// TwinCAT 3 PLC project Fs_Standard
// Title: FisoThemes Standard Library
// Company: FisoThemes
// ProjectVersion: 0.0.0.0
// ProgramVersion: 3.1.4023.0
// libraries:
//   Tc2_Standard, * (Beckhoff Automation GmbH)
//   Tc2_System, * (Beckhoff Automation GmbH)
//   Tc3_Module, * (Beckhoff Automation GmbH)
// project tree:
//   Core/DataUnitTypes/Alias/ FsT_Accessor.TcDUT, FsT_Char.TcDUT, FsT_SStr.TcDUT, FsT_MemArea.TcDUT, FsT_PlcAppInfo.TcDUT, FsT_PlcTaskInfo.TcDUT, FsT_Ptr.TcDUT, FsT_Size.TcDUT, FsT_Str.TcDUT, FsT_LStr.TcDUT, FsT_TypeClass.TcDUT, FsT_VarInfo.TcDUT
//   Core/DataUnitTypes/Enums/ FsE_Accessor.TcDUT
//   Core/DataUnitTypes/Structs/ FsST_PlcTaskInformation.TcDUT
//   Core/FunctionBlocks/ FsFB_Object.TcPOU, FsFB_ValueType.TcPOU
//   Core/Functions/ FsF_Cast.TcPOU, FsF_GetAddress.TcPOU, FsF_GetSize.TcPOU, FsF_GetPlcTaskInformation.TcPOU, FsF_GetTypeNameByAddress.TcPOU, FsF_GetTypeName.TcPOU, FsF_GetVariablePathByAddress.TcPOU, FsF_GetTypeNameByPath.TcPOU, FsF_GetVariablePath.TcPOU
//   Core/Interfaces/ FsI_Cloneable.TcIO, FsI_Equatable.TcIO, FsI_Unknown.TcIO, FsI_Object.TcIO, FsI_ValueType.TcIO
//   Core/Parameters/ FsParam_Core.TcGVL
//   Core/_Playground/ FsP_CorePlayground.TcPOU
//   ErrorHandling/DataUnitTypes/Alias/ FsT_ErrMsg.TcDUT, FsT_ErrSrc.TcDUT, FsT_ErrCode.TcDUT
//   ErrorHandling/FunctionBlocks/ FsFB_Error.TcPOU, FsFB_ErrorDefinition.TcPOU, FsFB_ErrorDefinitionOnInit.TcPOU
//   ErrorHandling/Functions/ FsF_Error.TcPOU, FsF_ErrorPath.TcPOU
//   ErrorHandling/Globals/ FsGVL_CodesysCmpErrors.TcGVL, FsGVL_ErrorCodes.TcGVL
//   ErrorHandling/Interfaces/ FsI_Error.TcIO
//   ErrorHandling/Parameters/ FsParam_ErrorHandling.TcGVL
//   / PlcTask.TcTTO
//   Project Information/ F_GetCompany.TcPOU, F_GetTitle.TcPOU, F_GetVersion.TcPOU
//   Version/ Global_Version.TcGVL
//   _Internal/FunctionBlocks/ FsFB_TcComIecApplicationInfo.TcPOU
//   _Internal/Globals/ _FsGVL.TcGVL
//   _Internal/ _MAIN.TcPOU
//   _TemplateFolder/_Playground/ FsP_TempPlayground.TcPOU
//   ErrorHandling/_Playground/ FsP_ErrorHandlingPlayground.TcPOU
// real-time tasks:
//   TASK PlcTask: cycle T#1ms, priority 20, ADS port 350

CONFIGURATION Fs_Standard
    RESOURCE PLC ON TwinCAT3
        TASK PlcTask(INTERVAL := T#1ms, PRIORITY := 20);
        PROGRAM _MAIN WITH PlcTask : _MAIN;
        PROGRAM FsP_CorePlayground WITH PlcTask : FsP_CorePlayground;
        PROGRAM FsP_ErrorHandlingPlayground WITH PlcTask : FsP_ErrorHandlingPlayground;
    END_RESOURCE
END_CONFIGURATION

// ---- Core/DataUnitTypes/Alias/FsT_Accessor.TcDUT
// An enum that can be used to represent getters and setters.
TYPE FsT_Accessor : FsE_Accessor; END_TYPE

// ---- Core/DataUnitTypes/Alias/FsT_Char.TcDUT
// Single character string.
TYPE FsT_Char : STRING(1); END_TYPE

// ---- Core/DataUnitTypes/Alias/FsT_SStr.TcDUT
// Short string.
// Size is a parameter located at FSParam_Core.nFST_SSTR_SIZE. | DEFAULT: 40
TYPE FsT_SStr : STRING(FSParam_Core.SSTR_SIZE); END_TYPE

// ---- Core/DataUnitTypes/Alias/FsT_MemArea.TcDUT
TYPE FsT_MemArea : Tc2_System.E_TcMemoryArea; END_TYPE

// ---- Core/DataUnitTypes/Alias/FsT_PlcAppInfo.TcDUT
TYPE FsT_PlcAppInfo : PlcAppSystemInfo; END_TYPE

// ---- Core/DataUnitTypes/Alias/FsT_PlcTaskInfo.TcDUT
TYPE FsT_PlcTaskInfo : FsST_PlcTaskInformation; END_TYPE

// ---- Core/DataUnitTypes/Alias/FsT_Ptr.TcDUT
TYPE FsT_Ptr : POINTER TO BYTE; END_TYPE

// ---- Core/DataUnitTypes/Alias/FsT_Size.TcDUT
TYPE FsT_Size : UXINT; END_TYPE

// ---- Core/DataUnitTypes/Alias/FsT_Str.TcDUT
// Standard FS string.
// Size is a parameter located at FSParam_Core.nFST_STR_SIZE. | DEFAULT: 80
TYPE FsT_Str : STRING(FSParam_Core.STR_SIZE); END_TYPE

// ---- Core/DataUnitTypes/Alias/FsT_LStr.TcDUT
// Long string.
// Size is a parameter located at FSParam_Core.nFST_STR_SIZE. | DEFAULT: 80
TYPE FsT_LStr : STRING(FSParam_Core.LSTR_SIZE); END_TYPE

// ---- Core/DataUnitTypes/Alias/FsT_TypeClass.TcDUT
TYPE FsT_TypeClass : __SYSTEM.TYPE_CLASS; END_TYPE

// ---- Core/DataUnitTypes/Alias/FsT_VarInfo.TcDUT
TYPE FsT_VarInfo : __SYSTEM.VAR_INFO; END_TYPE

// ---- Core/DataUnitTypes/Enums/FsE_Accessor.TcDUT
// An enum that can be used to represent getters and setters.
{attribute 'qualified_only'}
{attribute 'strict'}
{attribute 'to_string'}
TYPE FsE_Accessor :
(
	_ := 0,
	Get,
	Set
);
END_TYPE

// ---- Core/DataUnitTypes/Structs/FsST_PlcTaskInformation.TcDUT
TYPE FsST_PlcTaskInformation :
STRUCT
	 ObjId                   : OTCID; // Object ID of the task reference, from which the PLC program is called.
     CycleTime               : LTIME; // Task cycle time.
     Priority                : UINT; // Task priority.
     AdsPort                 : UINT; // Task ADS port.
     CycleCount              : UDINT; // Cycle counter. | NOTE: This refers to the actual system task and not to the task reference of the PLC project.
     DcTaskTime              : LINT; // Distributed Clock System Time. | NOTE: It remains constant for a task runtime.
     LastExecTime            : LTIME; // Cycle time required for the last cycle.
     FirstCycle              : BOOL; // During the first PLC task cycle, this variable has the value TRUE.
     CycleTimeExceeded       : BOOL; // Indicates whether the set task cycle time was exceeded.
     InCallAfterOutputUpdate : BOOL; // This TRUE if the origin of the current call is declared with the attribute 'TcCallAfterOutputUpdate'.
     RTViolation             : BOOL; // This variable has the value TRUE if the real-time limit is exceeded on a mixed core (Windows + real-time on one core).
     TaskName                : STRING(63); // Name of the task reference object in the PLC project (e.g. 'MyPlcProject_PlcTaskRef')
	 TaskIndex 				 : BYTE; // Task index of the task.
END_STRUCT
END_TYPE

// ---- ErrorHandling/DataUnitTypes/Alias/FsT_ErrMsg.TcDUT
TYPE FsT_ErrMsg : STRING(FsParam_ErrorHandling.ERROR_MSG_SIZE); END_TYPE

// ---- ErrorHandling/DataUnitTypes/Alias/FsT_ErrSrc.TcDUT
TYPE FsT_ErrSrc : STRING(FsParam_ErrorHandling.ERROR_SRC_SIZE); END_TYPE

// ---- ErrorHandling/DataUnitTypes/Alias/FsT_ErrCode.TcDUT
TYPE FsT_ErrCode : LINT; END_TYPE

// ---- Core/Parameters/FsParam_Core.TcGVL
{attribute 'qualified_only'}
VAR_GLOBAL CONSTANT
	STR_SIZE : FsT_Size := 80; // Size of general string.
	SSTR_SIZE : FsT_Size := 40; // Size of short string.
	LSTR_SIZE : FsT_Size := 255; // Size of long string.
	INFO_SCAN_SIZE : FsT_Size := 15000; // How many bytes to scan when looking for information. e.g. it's FsFB_Object to find the size of a child object in static memory.
END_VAR

// ---- ErrorHandling/Globals/FsGVL_CodesysCmpErrors.TcGVL
{attribute 'qualified_only'}
(* Error code are @ CmpErrors.Errors.<variable> from the CmpErrors2 Interfaces library.*)
VAR_GLOBAL CONSTANT
	ERR_OK 						: FsT_ErrCode := 16#0; 		//	Ok
	ERR_FAILED 					: FsT_ErrCode := 16#1; 		//	General error - To be used only for internal errors
	ERR_PARAMETER 				: FsT_ErrCode := 16#2; 		//	Invalid parameter for this operation
	ERR_NOTINITIALIZED 			: FsT_ErrCode := 16#3; 		//	Function cannot be executed, since component has not been initialized yet. It may work later, though
	ERR_VERSION 				: FsT_ErrCode := 16#4; 		//	Version conflict
	ERR_TIMEOUT 				: FsT_ErrCode := 16#5; 		//	Operation timed out
	ERR_NOBUFFER 				: FsT_ErrCode := 16#6; 		//	Insufficient memory to carry out the request
	ERR_PENDING 				: FsT_ErrCode := 16#A; 		//	For async-calls: call not complete, yet
	ERR_NUMPENDING 				: FsT_ErrCode := 16#B; 		//  Too many pending calls. Try later
	ERR_NOTIMPLEMENTED 			: FsT_ErrCode := 16#C; 		//  The function is not implemented
	ERR_INVALIDID 				: FsT_ErrCode := 16#D; 		//  No object with the provided id found
	ERR_OVERFLOW 				: FsT_ErrCode := 16#E; 		//	Integer overflow
	ERR_BUFFERSIZE 				: FsT_ErrCode := 16#F; 		//	The size of a buffer is too small OR invalid
	ERR_NO_OBJECT 				: FsT_ErrCode := 16#10;		//	No object with THIS specified name available
	ERR_NOMEMORY 				: FsT_ErrCode := 16#11;		//  No heap memory available
	ERR_DUPLICATE 				: FsT_ErrCode := 16#12A;  	//  An object with the same name is still available
	ERR_MEMORY_OVERWRITE 		: FsT_ErrCode := 16#13;  	//  Heap memory was written out of bounds! Memory overwrite error
	ERR_INVALID_HANDLE 			: FsT_ErrCode := 16#14;  	//  Invalid handle to an object
	ERR_END_OF_0BJECT 			: FsT_ErrCode := 16#15;  	//  End OF object reached
	ERR_NO_CHANGE 				: FsT_ErrCode := 16#16;  	//  No changes done
	ERR_INVALID_INTERFACE 		: FsT_ErrCode := 16#17;  	//  Invalid OR unknown interface
	ERR_NOT_SUPPORTED 			: FsT_ErrCode := 16#18;  	//  Functionality not supported
	ERR_NO_ACCESS_RIGHTS 		: FsT_ErrCode := 16#19;  	//  No access rights for this operation
	ERR_OUT_OF_LIMITS 			: FsT_ErrCode := 16#1A;  	//  Specified limits of a resource exceeded
	ERR_ENTRIES_REMAINING 		: FsT_ErrCode := 16#18;  	//  Remaining entries that could not be transmitted because of buffer limitation
	ERR_INVALID_SESSION_ID 		: FsT_ErrCode := 16#1C;  	//  Invalid online sessionid
	ERR_EXCEPTION 				: FsT_ErrCode := 16#1D;  	//  Exception occurred
	ERR_SIGNATURE_MISMATCH 		: FsT_ErrCode := 16#1E;		//	Signature mismatch of an api function
	ERR_VERSION_MISMATCH 		: FsT_ErrCode := 16#1F;		//	Version mismatch
	ERR_TYPE_MISMATCH 			: FsT_ErrCode := 16#20;		//	Type mismatch
	ERR_ID_MISMATCH 			: FsT_ErrCode := 16#21;		//	ID mismatch
	ERR_NO_CONSISTENCY 			: FsT_ErrCode := 16#22;		//	Consistency error
	ERR_NO_COMM_CYCLE 			: FsT_ErrCode := 16#23;		//	No COMM_CYCLE needed
	ERR_DONT_SUSPEND_TASK 		: FsT_ErrCode := 16#24;		//	Do not suspend task after an exception
	ERR_MEMORY_LOCK_FAILED 		: FsT_ErrCode := 16#25;		//	Memory cannot be locked in this operation
	ERR_LICENSE_MISSING 		: FsT_ErrCode := 16#26;		//	License missing for the runtime
	ERR_OPERATION_DENIED 		: FsT_ErrCode := 16#27;		//	Operation denied 
	ERR_DEVICE 					: FsT_ErrCode := 16#28;		//	Device error
	ERR_DISK_FULL 				: FsT_ErrCode := 16#29;		//	Disk full
	ERR_CRC_FAILED 				: FsT_ErrCode := 16#30;		//	Internal use in runtime
	ERR_MEDIA_ERASE 			: FsT_ErrCode := 16#31;		//	Internal use in runtime
	ERR_FILE_ERROR 				: FsT_ErrCode := 16#32;		//	File error. e.g. cannot open a file for writing because it could be write protected
	ERR_NO_RETAIN_MEMORY 		: FsT_ErrCode := 16#33;		//	No retain memory available
	ERR_OUT_OF_LIMITS_MIN 		: FsT_ErrCode := 16#34;		//	Specified minimum-limit of a resource exceeded
	ERR_OUT_OF_LIMITS_MAX 		: FsT_ErrCode := 16#35;		//	Specified maximum-limit of a resource exceeded
	ERR_SIZE_MISMATCH 			: FsT_ErrCode := 16#36;		//	Size mismatch
	ERR_CALL_AGAIN 				: FsT_ErrCode := 16#37;		//	Operation is not yet finished, call function again to proceed
	ERR_NOTHING_TO_DO 			: FsT_ErrCode := 16#38;		//	Operation has nothing to do. No execution.
	ERR_SECURITY_CHECKS_FAILED 	: FsT_ErrCode := 16#39;		//	Some security checks have failed. /* This is a generic error code to report this error over public channels. In this case the error code doesn’t provide a detailed cause for the error. */
	ERR_INVALID_SEQUENCE 		: FsT_ErrCode := 16#3A;		//	 
	ERR_INVALID_REFERENCE 		: FsT_ErrCode := 16#3B;		//	Dereferencing an IEC reference in IecVarAccess failed due TO invalid destination address, e. G. NULL.
	ERR_CONVERSION_INCOMPLETE 	: FsT_ErrCode := 16#3C;		//	Conversion of string encodings was not lossless.
	ERR_SOCK_NOTINITIALIZED 	: FsT_ErrCode := 16#201;   	//  Socket errors (range: 0x0200 - 0X02FF)
	ERR_SOCK_NOTSOCKET 			: FsT_ErrCode := 16#202;   	//  The provided socket handle is invalid
	ERR_SOCK_AFUNSUPPORTED 		: FsT_ErrCode := 16#203;   	//  The address family is not supported
	ERR_SOCK_PROTOUNSUPPORTED  	: FsT_ErrCode := 16#204;   	//  Protocol is not supported */
	ERR_SOCK_NOBUFFER 			: FsT_ErrCode := 16#205;   	//  Not enough buffer to handle the request */
	ERR_SOCK_WOULDBLOCK 		: FsT_ErrCode := 167206;   	//  Socket is in nonblocking mode but THIS call would block =/
	ERR_SOCK_ADDRINUSE 			: FsT_ErrCode := 16#207;   	//  The provided address is already in use */
	ERR_SOCK_ADDRNOTAVAILABLE  	: FsT_ErrCode := 16#208;   	//  The provided address is not available on THIS computer */
	ERR_SOCK_CONNREFUSED 		: FsT_ErrCode := 16#209;   	//  Connection has been refused by the remote host */
	ERR_SOCK_TIMEDOUT 			: FsT_ErrCode := 16#20A;   	//  Operation timed out */
	ERR_SOCK_HOSTNOTFOUND 		: FsT_ErrCode := 16#208;   	//  The host has NOT been found */
	ERR_SOCK_HOSTUNREACHABLE  	: FsT_ErrCode := 16#20C;   	//  Host is unreachable */
	ERR_SOCK_1SCONNECTED 		: FsT_ErrCode := 16#20D;   	//  Socket is already connected =/
	ERR_SOCK_NOTCONNECTED 		: FsT_ErrCode := 16#20E;   	//  The socket is not connected */
	ERR_SOCK_SHUTDOWN 			: FsT_ErrCode := 16#20F;   	//  Shutdown has been called on the socket =/
	ERR_SOCK_MSGSIZE 			: FsT_ErrCode := 16#210;   	//  FOR sockets of type DGRAM. The package to send exceeds the maximum package size =/
	ERR_SOCK_CLOSED 			: FsT_ErrCode := 167211;   	//  Socket has been gracefully closed. No more send/receives allowed =/
	ERR_L7_TAG_MISSING 			: FsT_ErrCode := 16#300;	//  Tag missing in online communication buffer
	ERR_L7_UNKNOWNCMDGROUP 		: FsT_ErrCode := 16#301;	//  Unknown command group
	ERR_L7_UNKNOWNCMD 			: FsT_ErrCode := 16#302;	//  Unknown command (within a valid command group)
	ERR_L7_INCOMPLETE 			: FsT_ErrCode := 16#303;	//  Level 7 service incomplete
END_VAR

// ---- ErrorHandling/Globals/FsGVL_ErrorCodes.TcGVL
{attribute 'qualified_only'}
VAR_GLOBAL CONSTANT
	NO_ERROR 			: FsT_ErrCode := 16#0; // No error.
	GENERAL 			: FsT_ErrCode := 16#1; // General error.
	INVALID_PARAMTERS 	: FsT_ErrCode := 16#2; // The paramters for this operation are invalid.
	TIMEDOUT 			: FsT_ErrCode := 16#3; // The operation took too long to complete.
	TYPE_MISMATCH 		: FsT_ErrCode := 16#4; // The wrong type is assigned to the variable or used in the expression.
	SIZE_MISMATCH 		: FsT_ErrCode := 16#5; // The size of two or more objects or values are not the same.
	INVALID_INTERFACE 	: FsT_ErrCode := 16#6; // The interface is null or invalid.
	MISSING_INTERFACE 	: FsT_ErrCode := 16#7; // The object does not implement the required interface.
	OUT_OF_BOUNDS 		: FsT_ErrCode := 16#8; // Attempted to access an element that is outside outside the valid range.
	OUT_OF_LIMITS 		: FsT_ErrCode := 16#9; // A value is outside of the valid range
END_VAR

// ---- ErrorHandling/Parameters/FsParam_ErrorHandling.TcGVL
{attribute 'qualified_only'}
VAR_GLOBAL CONSTANT
	ERROR_MSG_SIZE : FsT_Size := 255; // String length of error message.
	ERROR_SRC_SIZE : FsT_Size := 255; // String length of error source.
END_VAR

// ---- Version/Global_Version.TcGVL
{attribute 'TcGenerated'}
{attribute 'no-analysis'}
{attribute 'linkalways'}
// This function has been automatically generated from the project information.
VAR_GLOBAL CONSTANT
	{attribute 'const_non_replaced'}
	stLibVersion_FisoThemes_Standard_Library : ST_LibVersion := (iMajor := 0, iMinor := 0, iBuild := 0, iRevision := 0, nFlags := 0, sVersion := '0.0.0.0');
END_VAR

// ---- _Internal/Globals/_FsGVL.TcGVL
{attribute 'qualified_only'}
VAR_GLOBAL INTERNAL
END_VAR
VAR_GLOBAL CONSTANT INTERNAL
	fbTcComIecApplicationInfo : FsFB_TcComIecApplicationInfo := ();
END_VAR

// ---- Core/Interfaces/FsI_Cloneable.TcIO
// Generic interface for creating clones of objects.
INTERFACE FsI_Cloneable EXTENDS FsI_Unknown

// Returns a clone of the object that exits in dynamic memory.
// Clone must be freed from dynamic memory manually when done.
// A clone is an identical object that occupies a new memory space.
// References from the original object are shared.
METHOD Clone : FsI_Object
VAR_OUTPUT
	e : FsFB_Error;
END_VAR
END_METHOD

END_INTERFACE

// ---- Core/Interfaces/FsI_Equatable.TcIO
// Generic interface for cgecking objects for equality
INTERFACE FsI_Equatable EXTENDS FsI_Unknown

// Compares this object to another object and returns TRUE if they are equal, or FALSE otherwise.
METHOD Equals : BOOL
VAR_INPUT
	ipObject : FsI_Object;
END_VAR
VAR_OUTPUT
	e : FsFB_Error;
END_VAR
END_METHOD

END_INTERFACE

// ---- Core/Interfaces/FsI_Unknown.TcIO
// Root interface of all FS objects. 
// Inherits __SYSTEM.IQueryInterface which is used to query an object interface/pointer for one of its interfaces.
INTERFACE FsI_Unknown EXTENDS __SYSTEM.IQueryInterface

END_INTERFACE

// ---- Core/Interfaces/FsI_Object.TcIO
// Generic interface that defines the basic properties and methods of an object in the FisoThemes Standard Library.
INTERFACE FsI_Object EXTENDS FsI_Unknown

// Pointer to the object in memory.
PROPERTY Address : FsT_Ptr
GET
END_GET
END_PROPERTY

// Represents the path to the object.
PROPERTY InstancePath : FsT_LStr
GET
END_GET
END_PROPERTY

// Checks if the current object is the same as (reference-wise) object as the input object.
METHOD Is : BOOL
VAR_INPUT
	ipObject : FsI_Object;
END_VAR
END_METHOD

// Memory area that the object is allocated in.
PROPERTY MemoryArea : FsT_MemArea
GET
END_GET
END_PROPERTY

//  Size of the object in bytes.
PROPERTY Size : FsT_Size
GET
END_GET
END_PROPERTY

// Converts this object to a string representation.
METHOD ToString : FsT_LStr
END_METHOD

// A string that represents the type of the object.
PROPERTY TypeName : FsT_Str
GET
END_GET
END_PROPERTY

END_INTERFACE

// ---- Core/Interfaces/FsI_ValueType.TcIO
// Generic interface for assignable objects.
// FsI_Object contains the pragma {attribute 'no_assign'} to stop unsafe copies during upcasting.
// If an object can safely be assigned with the assignment operator ('='), using this interface. 
INTERFACE FsI_ValueType EXTENDS FsI_Object

END_INTERFACE

// ---- ErrorHandling/Interfaces/FsI_Error.TcIO
// General interface for error classes.
INTERFACE FsI_Error EXTENDS FsI_Unknown

PROPERTY Code : FsT_ErrCode
GET
END_GET
END_PROPERTY

PROPERTY Message : FsT_ErrMsg
GET
END_GET
END_PROPERTY

END_INTERFACE

// ---- _Internal/_MAIN.TcPOU
PROGRAM INTERNAL _MAIN
VAR
END_VAR

END_PROGRAM

// ---- Core/_Playground/FsP_CorePlayground.TcPOU
PROGRAM INTERNAL FsP_CorePlayground
VAR
	bStart, bGo: BOOL := TRUE;
	fbObj : FsFB_Object;
	rObj: REFERENCE TO FsFB_Object;
	fbErr : FsFB_Error;
	fbErr2 : FsFB_Error;
	arpData : ARRAY[0..3] OF FsT_Ptr;
	fbErrDef : FsFB_ErrorDefinitionOnInit(11, 'Dogs');
	Sz0,Sz1 : FsT_Size;
	sName : STRING(255);
	arData : ARRAY[0..3] OF FsT_LStr;
	
	ii : ITcUnknown;
	AppInfo : FsT_PlcAppInfo;
	TaskInfo : FsT_PlcTaskInfo;
	pCC : ULINT;
	hRes : HRESULT; 
END_VAR

arData[0] := fbObj.InstancePath;
arData[1] := fbObj.TypeName;
arData[2] := FsF_GetVariablePathByAddress(ADR(fbObj), SIZEOF(fbObj));
Sz0 := fbObj.Size;
rObj REF= fbErr;
FsF_Cast(rObj, fbErr2);
arpData[0] := ADR(fbErr);
arpData[1] := ADR(fbErr2);
AppInfo := TwinCAT_SystemInfoVarList._AppInfo;
TaskInfo :=  FsF_GetPlcTaskInformation();

END_PROGRAM

// ---- Core/FunctionBlocks/FsFB_Object.TcPOU
// Base class of all classes in the FisoThemes Standard Library.
{attribute 'enable_dynamic_creation'}
{attribute 'reflection'}
{attribute 'no_assign'}
{attribute 'no_explicit_call' := 'direct call for this function block is not allowed'} 
FUNCTION_BLOCK FsFB_Object IMPLEMENTS FsI_Object

// Private local variable to store object's size
METHOD PRIVATE _Size : FsT_Size
VAR_INPUT
	Accessor : FsT_Accessor;
	Data : FsT_Size;
END_VAR
VAR_INST
	Store : FsT_Size;
END_VAR
CASE Accessor OF
	FsT_Accessor.Set:
		_Size := Store := Data;
	FsT_Accessor.Get:
		_Size := Store;
	END_CASE
END_METHOD

// Pointer to the object in memory.
PROPERTY FINAL Address : FsT_Ptr
GET
Address := THIS;
END_GET
END_PROPERTY

// A string that represents the type of the object if the object is created dynamically.
// Classes indeed for dynamic use must override this property.
PROPERTY PROTECTED DynamicTypeName : FsT_Str
GET
DynamicTypeName := 'FsFB_Object';
END_GET
END_PROPERTY

{attribute 'hide'}
METHOD FB_init : BOOL
VAR_INPUT
	bInitRetains : BOOL; // if TRUE, the retain variables are initialized (warm start / cold start)
	bInCopyCode : BOOL;  // if TRUE, the instance afterwards gets moved into the copy code (online change)
END_VAR
VAR
	sTypeName : FsT_Str;
	i : FsT_Size := 0;
END_VAR
// If size has already been initialised then don't run this again.
IF THIS^.Size <> 0 THEN RETURN; END_IF

CASE THIS^.MemoryArea OF
// Attempt to get size of object.
	FsT_MemArea.Static:
	// If object in static memory try and look for it using the TcCOM object server and get it's size.
		FOR i := SIZEOF(THIS^) TO FsParam_Core.INFO_SCAN_SIZE DO
			sTypeName := FsF_GetTypeNameByAddress(THIS, i);
			IF sTypeName <> '' THEN EXIT; END_IF
			END_FOR
		THIS^._Size(FsT_Accessor.Set, i);
ELSE
// In any other case just return the base object size.
	THIS^._Size(FsT_Accessor.Set, SIZEOF(THIS^));
	END_CASE
END_METHOD

// Represents the path to the object.
PROPERTY FINAL InstancePath : FsT_LStr
GET
CASE THIS^.MemoryArea OF
	FsT_MemArea.Static: 
		InstancePath := FsF_GetVariablePathByAddress(THIS, THIS^.Size);
	FsT_MemArea.Dynamic:
		InstancePath := '<Dynamic>';
	FsT_MemArea.CNC:
		InstancePath := '<Unsupported>';
ELSE
	InstancePath := '<Unknown>';
	END_CASE
END_GET
END_PROPERTY

// Checks if the current object is the same as (reference-wise) object as the input object.
METHOD FINAL Is : BOOL
VAR_INPUT
	ipObject : FsI_Object;
END_VAR
IF ipObject <> 0 THEN Is := ipObject.Address = THIS; END_IF
END_METHOD

// Memory area that the object is allocated in.
PROPERTY FINAL MemoryArea : FsT_MemArea
GET
MemoryArea := Tc2_System.F_CheckMemoryArea(THIS, 1);
END_GET
END_PROPERTY

//  Size of the object in bytes.
PROPERTY Size : FsT_Size
GET
Size := THIS^._Size(FsT_Accessor.Get, 0);
END_GET
END_PROPERTY

// Converts this object to a string representation.
METHOD ToString : FsT_LStr
ToString := THIS^.TypeName;
END_METHOD

// A string that represents the type of the object.
PROPERTY FINAL TypeName : FsT_Str
GET
CASE THIS^.MemoryArea OF
	FsT_MemArea.Static: 
		TypeName := FsF_GetTypeNameByAddress(THIS, THIS^.Size);
	FsT_MemArea.Dynamic:
		TypeName := THIS^.DynamicTypeName;
	FsT_MemArea.CNC:
		TypeName := '<Unsupported>';
ELSE
	TypeName := '<Unknown>';
	END_CASE
END_GET
END_PROPERTY

END_FUNCTION_BLOCK

// ---- Core/Functions/FsF_GetTypeNameByAddress.TcPOU
// Returns the datatype of a variable as a string using its pointer and size.
// Variables allocated in dynamic memory are not supported.
FUNCTION FsF_GetTypeNameByAddress : FsT_Str
VAR_INPUT
	Address : FsT_Ptr; // Pointer to variable.
	Size : FsT_Size; // Size of variable in bytes.
END_VAR
VAR 
	nTmp : UDINT := SIZEOF(FsF_GetTypeNameByAddress);
END_VAR

_FsGVL.fbTcComIecApplicationInfo
	.GetInterface()
	.GetDatatypeNameByAddress(TO_UDINT(Size), Address, nTmp, ADR(FsF_GetTypeNameByAddress));

END_FUNCTION

// ---- Core/Functions/FsF_GetVariablePathByAddress.TcPOU
// Returns the name of a variable as a string using its pointer and size.
// Variables allocated in dynamic memory are not supported.
FUNCTION FsF_GetVariablePathByAddress : FsT_Str
VAR_INPUT
	Address : FsT_Ptr; // Pointer to variable.
	Size : FsT_Size; // Size of variable in bytes.
END_VAR
VAR
	nTmp : UDINT := SIZEOF(FsF_GetVariablePathByAddress);
END_VAR

_FsGVL.fbTcComIecApplicationInfo
	.GetInterface()
	.GetSymbolNameByAddress(TO_UDINT(Size), Address, nTmp, ADR(FsF_GetVariablePathByAddress));

END_FUNCTION

// ---- ErrorHandling/FunctionBlocks/FsFB_Error.TcPOU
// Base class for all error classes.
{attribute 'enable_dynamic_creation'}
{attribute 'reflection'}
{attribute 'no_explicit_call' := 'direct call for this function block is not allowed'}
FUNCTION_BLOCK FsFB_Error EXTENDS FsFB_ValueType IMPLEMENTS FsI_Error
VAR
	_Code : FsT_ErrCode := FsGVL_ErrorCodes.NO_ERROR;
	_Message : FsT_ErrMsg := 'No Error.';
END_VAR

PROPERTY Code : FsT_ErrCode
GET
Code := THIS^._Code;
END_GET
END_PROPERTY

PROPERTY PROTECTED DynamicTypeName : FsT_Str
GET
VAR
	fbVar : FsFB_Error;
	VarInfo : FsT_VarInfo := __VARINFO(fbVar); 
END_VAR
DynamicTypeName := VarInfo.TypeName;
END_GET
END_PROPERTY

PROPERTY Message : FsT_ErrSrc
GET
Message := THIS^._Message;
END_GET
END_PROPERTY

END_FUNCTION_BLOCK

// ---- Core/FunctionBlocks/FsFB_ValueType.TcPOU
// Base class for assignable objects.
// FsFB_Object contains the pragma {attribute 'no_assign'} to stop unsafe copies during upcasting.
// If an object can safely be assigned with the assignment operator ('='), using this interface. 
{attribute 'enable_dynamic_creation'}
{attribute 'reflection'}
{attribute 'no_explicit_call' := 'direct call for this function block is not allowed'} 
FUNCTION_BLOCK ABSTRACT FsFB_ValueType EXTENDS FsFB_Object IMPLEMENTS FsI_ValueType
VAR
END_VAR

PROPERTY PROTECTED DynamicTypeName : FsT_Str
GET
DynamicTypeName := 'FsFB_ValueType';
END_GET
END_PROPERTY

END_FUNCTION_BLOCK

// ---- ErrorHandling/FunctionBlocks/FsFB_ErrorDefinitionOnInit.TcPOU
// Function block for creating custom errors on initialisation.
{attribute 'enable_dynamic_creation'}
{attribute 'reflection'}
{attribute 'no_explicit_call' := 'direct call for this function block is not allowed'} 
FUNCTION_BLOCK FINAL FsFB_ErrorDefinitionOnInit EXTENDS FsFB_Error
VAR
END_VAR

PROPERTY PROTECTED DynamicTypeName : FsT_Str
GET
VAR
	fbVar : FsFB_ErrorDefinitionOnInit(0,'');
	VarInfo : FsT_VarInfo := __VARINFO(fbVar); 
END_VAR
DynamicTypeName := VarInfo.TypeName;
END_GET
END_PROPERTY

{attribute 'hide'}
METHOD FB_init : BOOL
VAR_INPUT
	bInitRetains : BOOL; // if TRUE, the retain variables are initialized (warm start / cold start)
	bInCopyCode : BOOL;  // if TRUE, the instance afterwards gets moved into the copy code (online change)
	Code : FsT_ErrCode;
	Message : FsT_ErrMsg;
END_VAR
THIS^._Code := Code;
THIS^._Message := Message;
END_METHOD

END_FUNCTION_BLOCK

// ---- Core/Functions/FsF_Cast.TcPOU
// Casts an object of that implements FsI_Object to another type of object.
FUNCTION FsF_Cast : REFERENCE TO FsFB_Error
VAR_INPUT
	ipFrom : FsI_Object;
	ipTo : FsI_Object;
END_VAR

IF ipFrom = 0 OR_ELSE ipTo = 0 THEN 
	FsF_Cast REF= FsF_Error(FsGVL_ErrorCodes.INVALID_INTERFACE, 'Null interface casting. You cannot cast to or from a null interface.');
	RETURN; 
	END_IF
	
IF ipFrom.Size <> ipTo.Size THEN
	FsF_Cast REF= FsF_Error(FsGVL_ErrorCodes.SIZE_MISMATCH, 'Size mismatch. The sizes of the casting entities do not match.');
	RETURN;
	END_IF
	
Tc2_System.MEMCPY(FsF_GetAddress(ipTo), FsF_GetAddress(ipFrom), TO_UDINT(ipFrom.Size));
FsF_Cast REF= FsF_Error(FsGVL_ErrorCodes.NO_ERROR, '');

END_FUNCTION

// ---- ErrorHandling/Functions/FsF_Error.TcPOU
// Takes two input parameters, Code and Message, and returns an FsFB_Error object.
FUNCTION FsF_Error : REFERENCE TO FsFB_Error
VAR_INPUT
	Code : FsT_ErrCode;
	Message : FsT_ErrMsg;
END_VAR
VAR_STAT
	fbError : FsFB_ErrorDefinition;
END_VAR

CASE Code OF
	FsGVL_ErrorCodes.NO_ERROR: 
		fbError.Code := FsGVL_ErrorCodes.NO_ERROR;
		fbError.Message := 'No Error.';
ELSE
	fbError.Code :=	Code;
	fbError.Message := Message;
	END_CASE
FsF_Error REF= fbError;

END_FUNCTION

// ---- ErrorHandling/FunctionBlocks/FsFB_ErrorDefinition.TcPOU
// Function block for creating custom errors.
{attribute 'enable_dynamic_creation'}
{attribute 'reflection'}
{attribute 'no_explicit_call' := 'direct call for this function block is not allowed'} 
FUNCTION_BLOCK FINAL FsFB_ErrorDefinition EXTENDS FsFB_Error
VAR
END_VAR

PROPERTY Code : FsT_ErrCode
SET
THIS^._Code := Code;
END_SET
END_PROPERTY

PROPERTY PROTECTED DynamicTypeName : FsT_Str
GET
VAR
	fbVar : FsFB_ErrorDefinition;
	VarInfo : FsT_VarInfo := __VARINFO(fbVar); 
END_VAR
DynamicTypeName := VarInfo.TypeName;
END_GET
END_PROPERTY

PROPERTY Message : FsT_ErrSrc
SET
THIS^._Message := Message;
END_SET
END_PROPERTY

END_FUNCTION_BLOCK

// ---- Core/Functions/FsF_GetAddress.TcPOU
// Gets the address of an object from it's interface.
// Interface must extend FsI_Unknown.
FUNCTION FsF_GetAddress : FsT_Ptr
VAR_INPUT
	ipInterface : FsI_Unknown;
END_VAR
VAR
	pInterface : POINTER TO FsT_Ptr := ADR(ipInterface);
END_VAR

IF ipInterface = 0 THEN RETURN; END_IF
FsF_GetAddress := pInterface^ - SIZEOF(ipInterface);

END_FUNCTION

// ---- Core/Functions/FsF_GetPlcTaskInformation.TcPOU
FUNCTION FsF_GetPlcTaskInformation : FsT_PlcTaskInfo
VAR
	fbGetCurrentTaskIndex : GETCURTASKINDEX;
	PlcTaskSysInfo : PlcTaskSystemInfo;
	PlcTaskInformation:FsT_PlcTaskInfo;
END_VAR

fbGetCurrentTaskIndex();
PlcTaskSysInfo := TwinCAT_SystemInfoVarList._TaskInfo[fbGetCurrentTaskIndex.Index];
FsF_GetPlcTaskInformation.AdsPort 					:= PlcTaskSysInfo.AdsPort;
FsF_GetPlcTaskInformation.CycleCount 				:= PlcTaskSysInfo.CycleCount;
FsF_GetPlcTaskInformation.CycleTime 				:= TO_LTIME(PlcTaskSysInfo.CycleTime*100);
FsF_GetPlcTaskInformation.CycleTimeExceeded 		:= PlcTaskSysInfo.CycleTimeExceeded;
FsF_GetPlcTaskInformation.DcTaskTime 				:= PlcTaskSysInfo.DcTaskTime;
FsF_GetPlcTaskInformation.FirstCycle				:= PlcTaskSysInfo.FirstCycle;
FsF_GetPlcTaskInformation.InCallAfterOutputUpdate 	:= PlcTaskSysInfo.InCallAfterOutputUpdate;
FsF_GetPlcTaskInformation.LastExecTime 				:= TO_LTIME(PlcTaskSysInfo.LastExecTime*100);
FsF_GetPlcTaskInformation.ObjId 					:= PlcTaskSysInfo.ObjId;
FsF_GetPlcTaskInformation.Priority 					:= PlcTaskSysInfo.Priority;
FsF_GetPlcTaskInformation.RTViolation 				:= PlcTaskSysInfo.RTViolation;
FsF_GetPlcTaskInformation.TaskName 					:= PlcTaskSysInfo.TaskName;
FsF_GetPlcTaskInformation.TaskIndex 				:= fbGetCurrentTaskIndex.Index;

END_FUNCTION

// ---- ErrorHandling/_Playground/FsP_ErrorHandlingPlayground.TcPOU
PROGRAM INTERNAL FsP_ErrorHandlingPlayground
VAR
	bStart, bDestroy : BOOL;
	pObj, pObj2 : POINTER TO FsFB_ErrorDefinition;
	fbNoError : FsFB_Error;
	fbErrDef : FsFB_ErrorDefinitionOnInit(11, 'Dogs');
	MemArea : FsT_MemArea;
	ipUnk : FsI_Unknown;
	ipObj : FsI_Object;
	pItfs : POINTER TO ARRAY[0..6] OF FsT_Ptr;
	nData, nData2 : FsT_Size;
	sdata : FsT_LStr;
	TaskInfo : FsT_PlcTaskInfo;
END_VAR

fbNoError := fbErrDef;
sData := fbNoError.Message;
fbNoError := FsF_ErrorPath(11,'Cats', ipObj);
sdata := FsF_Error(11,'Cats').Message;
ipUnk := fbNoError;
ipObj := fbNoError;
pItfs := ADR(ipUnk);
pObj2 := ADR(fbNoError);
nData := SIZEOF(fbNoError);
nData2 := FsF_GetSize(ipObj);
TaskInfo :=  FsF_GetPlcTaskInformation();
IF bStart THEN 
	bStart := FALSE;
	pObj := __NEW(FsFB_ErrorDefinition);
	sData := pObj^.TypeName;
	END_IF
IF bDestroy THEN
	bDestroy := FALSE; 
	__DELETE(pObj);
	END_IF

END_PROGRAM

// ---- ErrorHandling/Functions/FsF_ErrorPath.TcPOU
// Returns an FsFB_Error object who's message includes the instance path of the object.
FUNCTION FsF_ErrorPath : REFERENCE TO FsFB_Error
VAR_INPUT
	Code : FsT_ErrCode;
	Message : FsT_ErrMsg;
	ipObject : FsI_Object;
END_VAR
VAR_STAT
	fbError : FsFB_ErrorDefinition;
END_VAR

IF ipObject = 0 THEN FsF_ErrorPath REF= FsF_Error(Code, Message); RETURN; END_IF
CASE Code OF
	FsGVL_ErrorCodes.NO_ERROR: 
		fbError.Code := FsGVL_ErrorCodes.NO_ERROR;
		fbError.Message := 'No Error.';
ELSE
	fbError.Code :=	Code;
	fbError.Message := Message;
	END_CASE
fbError.Message := CONCAT(fbError.Message, CONCAT(' | Path: ',ipObject.InstancePath));
FsF_ErrorPath REF= fbError;

END_FUNCTION

// ---- Core/Functions/FsF_GetSize.TcPOU
// Gets the size of an object in static memory via its interface.
// Interface must extend FsI_Unknown.
// NOTE: This is performance intensive. Cyclic use is not recommened.
FUNCTION FsF_GetSize : FsT_Size
VAR_INPUT
	ipInterface : FsI_Unknown;
END_VAR
VAR
	pAddress : FsT_Ptr;
END_VAR

pAddress := FsF_GetAddress(ipInterface);
IF pAddress = 0 THEN RETURN; END_IF
CASE Tc2_System.F_CheckMemoryArea(pAddress, 1) OF
	FsT_MemArea.Static:
		FOR FsF_GetSize := SIZEOF(ipInterface) TO FsParam_Core.INFO_SCAN_SIZE DO
			IF FsF_GetTypeNameByAddress(pAddress, FsF_GetSize) <> '' THEN RETURN; END_IF
			END_FOR
		FsF_GetSize := 0;
	END_CASE

END_FUNCTION

// ---- _Internal/FunctionBlocks/FsFB_TcComIecApplicationInfo.TcPOU
// Internal class that manages the ITcIecApplicationInfo TcCOM Interface used by Fs_Standard.
{attribute 'no_assign'}
{attribute 'no_explicit_call' := 'direct call for this function block is not allowed'} 
FUNCTION_BLOCK INTERNAL FINAL FsFB_TcComIecApplicationInfo IMPLEMENTS FsI_UnKnown
VAR
	_ipIecApplicationInformation : ITcIecApplicationInfo;
	_hIecApplicationInformation : HRESULT := Tc3_Module.GVL.E_FAIL;
END_VAR

{attribute 'hide'}
METHOD FB_exit : BOOL
VAR_INPUT
	bInCopyCode : BOOL; // if TRUE, the exit method is called for exiting an instance that is copied afterwards (online change).
END_VAR
// no online change
IF NOT bInCopyCode THEN
	// Safe release of ITcIecApplicationInfo.
    Tc3_Module.FW_SafeRelease(ADR(THIS^._ipIecApplicationInformation));
	THIS^._hIecApplicationInformation := Tc3_Module.GVL.E_FAIL;
	END_IF
END_METHOD

{attribute 'hide'}
{attribute 'no_explicit_call' := 'direct call for this method is not allowed'}
METHOD FB_init : BOOL
VAR_INPUT
	bInitRetains : BOOL; // if TRUE, the retain variables are initialized (warm start / cold start)
	bInCopyCode : BOOL;  // if TRUE, the instance afterwards gets moved into the copy code (online change)
END_VAR
// No online change.
IF NOT bInCopyCode THEN
	// Get instance of ITcIecApplicationInfo.
	THIS^._hIecApplicationInformation := Tc3_Module.FW_ObjMgr_GetObjectInstance(
		TwinCAT_SystemInfoVarList._AppInfo.ObjId, 
		TC_GLOBAL_IID_LIST.IID_ITcIecApplicationInfo, 
		ADR(THIS^._ipIecApplicationInformation)
	);
	END_IF
END_METHOD

METHOD GetInterface : ITcIecApplicationInfo
VAR_OUTPUT
	bSuccess : BOOL;
END_VAR
// If instance of ITcIecApplicationInfo failed to be obtained on 
// FB_init or FB_exit was explicitly called try to get it gain.
IF Tc3_Module.FAILED(THIS^._hIecApplicationInformation) THEN
	THIS^._hIecApplicationInformation := Tc3_Module.FW_ObjMgr_GetObjectInstance(
		TwinCAT_SystemInfoVarList._AppInfo.ObjId, 
		TC_GLOBAL_IID_LIST.IID_ITcIecApplicationInfo, 
		ADR(THIS^._ipIecApplicationInformation)
	);
	END_IF
	
bSuccess := Tc3_Module.SUCCEEDED(THIS^._hIecApplicationInformation);
GetInterface := THIS^._ipIecApplicationInformation;
END_METHOD

END_FUNCTION_BLOCK

// ---- Core/Functions/FsF_GetTypeName.TcPOU
// Returns the datatype of a variable as a string using its pointer and size.
// Variables allocated in dynamic memory are not supported.
FUNCTION FsF_GetTypeName : FsT_Str
VAR_INPUT
	Variable : ANY;
END_VAR
VAR 
	nTmp : UDINT := SIZEOF(FsF_GetTypeName);
END_VAR

_FsGVL.fbTcComIecApplicationInfo
	.GetInterface()
	.GetDatatypeNameByAddress(TO_UDINT(Variable.diSize), Variable.pValue, nTmp, ADR(FsF_GetTypeName));

END_FUNCTION

// ---- Core/Functions/FsF_GetTypeNameByPath.TcPOU
// Returns the datatype of a variable as a string using its path.
FUNCTION FsF_GetTypeNameByPath : FsT_Str
VAR_INPUT
	Path : FsT_LStr; // Variable/Symbol path as string | e.g. 'MAIN.nVar'
END_VAR
VAR 
	nTmp : UDINT := SIZEOF(FsF_GetTypeNameByPath);
END_VAR

_FsGVL.fbTcComIecApplicationInfo
	.GetInterface()
	.GetSymbolDatatype(Path, nTmp, ADR(FsF_GetTypeNameByPath));

END_FUNCTION

// ---- Core/Functions/FsF_GetVariablePath.TcPOU
// Returns the name of a variable as a string using its pointer and size.
// Variables allocated in dynamic memory are not supported.
FUNCTION FsF_GetVariablePath : FsT_Str
VAR_INPUT
	Variable : ANY;
END_VAR
VAR
	nTmp : UDINT := SIZEOF(FsF_GetVariablePath);
END_VAR

_FsGVL.fbTcComIecApplicationInfo
	.GetInterface()
	.GetSymbolNameByAddress(TO_UDINT(Variable.diSize), Variable.pValue, nTmp, ADR(FsF_GetVariablePath));

END_FUNCTION

// ---- Project Information/F_GetCompany.TcPOU
// This function has been automatically generated from the project information.
{attribute 'signature_flag' := '1073741824'}
{attribute 'TcGenerated'}
{attribute 'no-analysis'}
FUNCTION F_GetCompany : WSTRING
VAR_INPUT
	
END_VAR

F_GetCompany := "FisoThemes";

END_FUNCTION

// ---- Project Information/F_GetTitle.TcPOU
// This function has been automatically generated from the project information.
{attribute 'signature_flag' := '1073741824'}
{attribute 'TcGenerated'}
{attribute 'no-analysis'}
FUNCTION F_GetTitle : WSTRING
VAR_INPUT
	
END_VAR

F_GetTitle := "FisoThemes Standard Library";

END_FUNCTION

// ---- Project Information/F_GetVersion.TcPOU
// This function has been automatically generated from the project information.
{attribute 'signature_flag' := '1073741824'}
{attribute 'TcGenerated'}
{attribute 'no-analysis'}
FUNCTION F_GetVersion : ST_LibVersion
VAR_INPUT
	
END_VAR

F_GetVersion.iMajor := 0;
F_GetVersion.iMinor := 0;
F_GetVersion.iBuild := 0;
F_GetVersion.iRevision := 0;

END_FUNCTION

// ---- _TemplateFolder/_Playground/FsP_TempPlayground.TcPOU
PROGRAM INTERNAL FsP_TempPlayground
VAR
END_VAR

ObjectPlayground();

METHOD PRIVATE TempPlayground
VAR_STAT
END_VAR
END_METHOD

END_PROGRAM
